// TIA Portal V20 export
TYPE "LCFL_typeMaintenanceSiemens"
TITLE = HMI data for LCFL_Maintenance
// HMI data for LCFL_Maintenance
   STRUCT
      mtpData : "LCFL_typeMTPOSLevel";
      maintenance : "LCFL_typeMaintenance";
      enabled { ExternalWritable := 'False'} : Bool := FALSE;   // Funktionalität des Steuerelements ist aktiviert / Functionality of control module is enabled
   END_STRUCT;
END_TYPE
